FUNCTION_BLOCK Filtersample IMPLEMENTS ITFBASE
VAR_INPUT
END_VAR
VAR_OUTPUT
END_VAR
VAR
END_VAR

METHOD Clear : I_ITF1
VAR_INPUT
END_VAR
END_METHOD

METHOD METH1 : I_ITF1
VAR_INPUT
END_VAR
END_METHOD

PROPERTY Prop1 : I_ITF2
GET
END_GET
SET
END_SET
END_PROPERTY

END_FUNCTION_BLOCK

(* stored: Version 1.1.0.1, ProductVersion 3.1.4024.12
   POU Filtersample: Id {41f9b86b-a8e4-419b-84f6-e2bb7e5b82de}, SpecialFunc None
   Method Clear: Id {87982b53-d10a-479d-b733-38c8cc0d07f0}
   Method METH1: Id {46144ff5-86f6-43ed-9b50-6b1cc14274d3}
   Property Prop1: Id {17347acb-1eb9-4a92-b800-3b0cee382971}
   Get Get: Id {52b08e44-6b29-4faf-870e-56fd857ed7b7}
   Set Set: Id {f9b49df6-5433-44b2-8495-2a24e73748e6} *)
